# EPICS substitutions: apps/bomApp/Db/bom_channels.substitutions
file "db/bom_channel.template" {
pattern { P R CScode Counts }
{ bom_sc_ai_ 0 0 0 }
}
#{ bom_sc_ai_ 1 0 1 }
#{ bom_sc_ai_ 2 0 2 }
#{ bom_sc_ai_ 3 0 3 }
#{ bom_sc_ai_ 4 0 4 }
#{ bom_sc_ai_ 5 0 5 }
#{ bom_sc_ai_ 6 0 6 }
#{ bom_sc_ai_ 7 0 7 }
#{ bom_sc_ai_ 8 0 8 }
#{ bom_sc_ai_ 9 0 9 }
#{ bom_sc_ai_ 10 0 10 }
#{ bom_sc_ai_ 11 0 11 }
#{ bom_sc_ai_ 12 0 12 }
#{ bom_sc_ai_ 13 0 13 }
#{ bom_sc_ai_ 14 0 14 }
#{ bom_sc_ai_ 15 0 15 }
#}
#
